# EPICS autosave request: iocBoot/sioc-li14-im01/sioc-li14-im01.req
file "facet2.req" AREA=LI14,POS=890
